{attribute 'qualified_only'}
VAR_GLOBAL
	bAuto 		: BOOL;
	bManuel 	: BOOL;
	bRunning 	: BOOL;
END_VAR

(* stored: Version 1.1.0.1
   GVL G_Mode: Id {cef963f9-2807-4386-8502-cf4081ad3059} *)
